Fanuc KAREL source: f_hand2_t.kl

PROGRAM F_HAND2_T
VAR i : INTEGER
  b : BOOLEAN
BEGIN
    CLOSE HAND 1
    RELAX HAND 2
    OPEN HAND 5
    OPEN HAND i
    CLOSE HAND i+1
    DOUT[3] = TRUE
    b = DOUT[3]
END F_HAND2_T
